Staubli VAL3: orderZone.pgx

program orderZone(num x_nDistance (dimensions=1), num x_nType (dimensions=1), num x_nTrajectory (dimensions=1), num& x_nBest[] (dimensions=1))
  local num l_nValue[4]
  local num i
  local bool l_bFound
begin
  //
  // check if the new HOME trajectory is better then the last one...
  //
  // MOVETYPE PRIORITY
  //
  // BOX -> SPHERE -> PLANE
  //
  // SAME MOVETYPE
  //
  // check the distance from the plane or the center of the sphere
  //
  // x_nTrajectory= home index
  // 0= joint index
  // x_nDistance= nDistance
  // type CUBE-SPHERE-PLANE= nCoeff
  //
  // copy all the value
  l_nValue=x_nTrajectory
  l_nValue[1]=0
  l_nValue[2]=x_nDistance
  l_nValue[3]=x_nType
  // order all
  // MINOR
  if x_nType<nCoeff
    // insert into
    call insertValue(l_nValue,0)
    // EQUAL order by distance
  elseIf x_nType==nCoeff
    // order by distance
    for i=0 to size(nCoeff)-1
      if x_nDistance<=nDistance[i] or i==size(nCoeff)-1
        // insert
        call insertValue(l_nValue,i)
        // exit
        i=size(nCoeff)-1
      endIf
    endFor
    // MAJOR
  elseIf x_nType>nCoeff
    // order by type
    for i=0 to size(nCoeff)-1
      if nCoeff[i]==x_nType
        // found it
        l_bFound=true
        if x_nDistance<=nDistance[i] or i==size(nCoeff)-1
          // insert
          call insertValue(l_nValue,i+1)
          // exit
          i=size(nCoeff)-1
        endIf
        // not the same but the prevoius one was ok
      elseIf l_bFound
        // insert one before
        call insertValue(l_nValue,i)
        // exit
        i=size(nCoeff)-1
        // found in the last item
      elseIf x_nDistance<=nDistance[i] or (i==size(nCoeff)-1)
        if nDistance[0]==-1
          // first item
          call insertValue(l_nValue,i)
        else
          // insert
          call insertValue(l_nValue,i+1)
        endIf
        // exit
        i=size(nCoeff)-1
      endIf
    endFor
  endIf
end
